{attribute 'linkalways'} 
{attribute 'no_explicit_call' := 'This FB is a CLASS and must be accessed using methods or properties'}
{attribute 'enable_dynamic_creation'}
FUNCTION_BLOCK _ETcVnAdaptiveThresholdMethod EXTENDS EnumDatatypeBase
VAR
	localData : ETcVnAdaptiveThresholdMethod;
	activeData : REFERENCE TO ETcVnAdaptiveThresholdMethod;
	enumBaseDatatype : _DINT(localData);
END_VAR

METHOD PRIVATE AddLocalEnumeration
VAR_INPUT
	Enumeration : T_MAXSTRING;
	Value : ETcVnAdaptiveThresholdMethod;
END_VAR
AddEnumeration(Enumeration, Value);
END_METHOD

PROPERTY PUBLIC Address : PVOID
GET
Address := ADR(activeData);
END_GET
END_PROPERTY

METHOD PUBLIC ClearReference
VAR_INPUT
END_VAR
activeData REF= localData;
SetBaseDatatypeReference();
END_METHOD

METHOD PUBLIC Clone : I_Datatype
VAR
    pClone : POINTER TO _ETcVnAdaptiveThresholdMethod;
END_VAR
pClone := __NEW(_ETcVnAdaptiveThresholdMethod(InitialValue := Value));
Clone := pClone^;
END_METHOD

METHOD FB_init : BOOL
VAR_INPUT
	bInitRetains : BOOL; // if TRUE, the retain variables are initialized (warm start / cold start)
	bInCopyCode : BOOL;  // if TRUE, the instance afterwards gets moved into the copy code (online change)
	InitialValue : ETcVnAdaptiveThresholdMethod;
END_VAR
localData := InitialValue;
AddBaseDatatype(enumBaseDatatype);
ClearReference();

AddLocalEnumeration('TCVN_ATM_MEAN', ETcVnAdaptiveThresholdMethod.TCVN_ATM_MEAN);
AddLocalEnumeration('TCVN_ATM_GAUSSIAN', ETcVnAdaptiveThresholdMethod.TCVN_ATM_GAUSSIAN);
END_METHOD

PROPERTY PUBLIC Identifier : T_MAXSTRING
GET
Identifier := 'ETcVnAdaptiveThresholdMethod';
END_GET
END_PROPERTY

METHOD IsEnumeratorValueEqual : BOOL
VAR_INPUT
	Enumerator : I_KeyValueForwardEnumerator;
END_VAR
VAR
	storedValue : ETcVnAdaptiveThresholdMethod;
END_VAR
IF NOT Enumerator.TryGet(storedValue) THEN
	RETURN;
END_IF

IsEnumeratorValueEqual := storedValue = activeData;
END_METHOD

METHOD PUBLIC MakeReferenceTo
VAR_INPUT
	ReferenceTarget : REFERENCE TO ETcVnAdaptiveThresholdMethod;
END_VAR
activeData REF= ReferenceTarget;
SetBaseDatatypeReference();
END_METHOD

METHOD PROTECTED SetBaseDatatypeReference
VAR_INPUT
END_VAR
enumBaseDatatype.MakeReferenceTo(activeData);
END_METHOD

PROPERTY PUBLIC Size : UDINT
GET
Size := SIZEOF(activeData);
END_GET
END_PROPERTY

METHOD TryMakeReferenceTo : BOOL
VAR_INPUT
	Target : I_Datatype;
END_VAR
VAR
	targetAsEnum : I_EnumDatatype;
	pTargetData : POINTER TO ETcVnAdaptiveThresholdMethod;
END_VAR
IF NOT Target.TryResolveAsEnumDatatype(targetAsEnum) THEN
	RETURN;
END_IF

IF targetAsEnum.Identifier <> Identifier THEN
	RETURN;
END_IF

pTargetData := Target.Address;
activeData REF= pTargetData^;
SetBaseDatatypeReference();
TryMakeReferenceTo := TRUE;
END_METHOD

PROPERTY PUBLIC Value : ETcVnAdaptiveThresholdMethod
GET
Value := activeData;
END_GET
SET
activeData := Value;
END_SET
END_PROPERTY

END_FUNCTION_BLOCK

(* stored: Version 1.1.0.1
   POU _ETcVnAdaptiveThresholdMethod: Id {26a3241b-78b8-02fb-127a-34cd31b93f52}, SpecialFunc None
   Folder Constructor: Id {c1f7c7ee-1cd0-0062-0d38-995e27dd0240}
   Folder Private: Id {d7cf7516-76db-09db-0558-887c95dcf8b5}
   Folder Protected: Id {b6d8bef6-5508-007f-1870-d4045cb53871}
   Method AddLocalEnumeration: Id {87a0d2e2-7d81-093c-19cc-ad6e23d940f2}
   Property Address: Id {c6336590-9e3e-02d5-22c5-90e4e73b79ba}
   Get Get: Id {48342524-9c19-0ef3-3379-204e26665ddb}
   Method ClearReference: Id {20da2f1a-840d-0cef-3ef1-ea9161bc08d8}
   Method Clone: Id {950cce9b-c0f0-01a2-1d7d-b16c0f4da112}
   Method FB_init: Id {ef58a7c0-dc3b-0802-301a-0bcd1c6453c2}
   Property Identifier: Id {e261b1e0-5408-0619-0a9b-da6a7e993265}
   Get Get: Id {4690aae6-c85f-0b58-00bc-281fccf4af28}
   Method IsEnumeratorValueEqual: Id {eafc55bd-b709-0689-03a9-4d6575259f9d}
   Method MakeReferenceTo: Id {8f309036-fbdf-0162-325f-a8d1c0edd9c3}
   Method SetBaseDatatypeReference: Id {76344340-d5b9-09f6-0c2e-bb98b5a474f5}
   Property Size: Id {621d2e0c-d20e-059b-0d89-e95ba9247fa0}
   Get Get: Id {58079bac-7cca-0ecf-0f70-cc349d3ea793}
   Method TryMakeReferenceTo: Id {69a76e1c-1af8-00b2-2032-2c34c2e227e9}
   Property Value: Id {3ccf15d2-b3b1-05f0-275c-7e6c44b41f81}
   Get Get: Id {bbce4832-dd75-0ca4-00e3-8deb6882c580}
   Set Set: Id {ed7a38f1-0a73-047d-1fae-0c2e83904170} *)
